// TIA Portal V17 program export: 1 tag tables, 0 data types, 18 data blocks, 11 code blocks (in call order from the OBs), 0 instance data blocks

VAR_GLOBAL   // PLC tag table "默认变量表"
   "1号计量泵运行" AT %I0.0 : Bool;
   "2号计量泵运行" AT %I0.2 : Bool;
   "3号计量泵运行" AT %I0.4 : Bool;
   "1号计量泵故障" AT %I0.1 : Bool;
   "2号计量泵故障" AT %I0.3 : Bool;
   "3号计量泵故障" AT %I0.5 : Bool;
   "1号药池电动阀开到位" AT %I0.6 : Bool;
   "2号药池电动阀开到位" AT %I1.0 : Bool;
   "1号药池电动阀关到位" AT %I0.7 : Bool;
   "2号药池电动阀关到位" AT %I1.1 : Bool;
   新旧电柜控制切换 AT %I1.2 : Bool;
   本电柜和中控控制切换 AT %I1.3 : Bool;
   "1号计量泵启停" AT %Q0.0 : Bool;
   "2号计量泵启停" AT %Q0.1 : Bool;
   "3号计量泵启停" AT %Q0.2 : Bool;
   "1号药池电动阀打开关闭" AT %Q0.3 : Bool;
   "2号药池电动阀打开关闭" AT %Q0.4 : Bool;
END_VAR

DATA_BLOCK "RS-485流量计1"
{ S7_Optimized_Access := 'FALSE' }
VERSION : 0.1
NON_RETAIN
   STRUCT 
      "40001" : Word;
      "40002" : Word;
      "40003" : Word;
      "40004" : Word;
      "40005" : Word;
      "40006" : Word;
      "40007" : Word;
      "40008" : Word;
      "40009" : Word;
      "40010" : Word;
      "40011" : Word;
      "40012" : Word;
      "40013" : Word;
      "40014" : Word;
      "40015" : Word;
      "40016" : Word;
      "40017" : Word;
      "40018" : Word;
      "40019" : Word;
      "40020" : Word;
      "40021" : Word;
      "40022" : Word;
      "40023" : Word;
      "40024" : Word;
      "40025" : Word;
      "40026" : Word;
      "40027" : Word;
      "40028" : Word;
      "40029" : Word;
      "40030" : Word;
      "40031" : Word;
      "40032" : Word;
      "40033" : Word;
      "40034" : Word;
      "40035" : Word;
      "40036" : Word;
      "40037" : Word;
      "40038" : Word;
      "40039" : Word;
      "40040" : Word;
      "40041" : Word;
      "40042" : Word;
      "40043" : Word;
      "40044" : Word;
      "40045" : Word;
      "40046" : Word;
      "40047" : Word;
      "40048" : Word;
      "40049" : Word;
      "40050" : Word;
   END_STRUCT;


BEGIN

END_DATA_BLOCK

DATA_BLOCK "RS-485流量计2"
{ S7_Optimized_Access := 'FALSE' }
VERSION : 0.1
NON_RETAIN
   STRUCT 
      "40001" : Word;
      "40002" : Word;
      "40003" : Word;
      "40004" : Word;
      "40005" : Word;
      "40006" : Word;
      "40007" : Word;
      "40008" : Word;
      "40009" : Word;
      "40010" : Word;
      "40011" : Word;
      "40012" : Word;
      "40013" : Word;
      "40014" : Word;
      "40015" : Word;
      "40016" : Word;
      "40017" : Word;
      "40018" : Word;
      "40019" : Word;
      "40020" : Word;
      "40021" : Word;
      "40022" : Word;
      "40023" : Word;
      "40024" : Word;
      "40025" : Word;
      "40026" : Word;
      "40027" : Word;
      "40028" : Word;
      "40029" : Word;
      "40030" : Word;
      "40031" : Word;
      "40032" : Word;
      "40033" : Word;
      "40034" : Word;
      "40035" : Word;
      "40036" : Word;
      "40037" : Word;
      "40038" : Word;
      "40039" : Word;
      "40040" : Word;
      "40041" : Word;
      "40042" : Word;
      "40043" : Word;
      "40044" : Word;
      "40045" : Word;
      "40046" : Word;
      "40047" : Word;
      "40048" : Word;
      "40049" : Word;
      "40050" : Word;
   END_STRUCT;


BEGIN

END_DATA_BLOCK

DATA_BLOCK "RS-485流量计3"
{ S7_Optimized_Access := 'FALSE' }
VERSION : 0.1
NON_RETAIN
   STRUCT 
      "40001" : Word;
      "40002" : Word;
      "40003" : Word;
      "40004" : Word;
      "40005" : Word;
      "40006" : Word;
      "40007" : Word;
      "40008" : Word;
      "40009" : Word;
      "40010" : Word;
      "40011" : Word;
      "40012" : Word;
      "40013" : Word;
      "40014" : Word;
      "40015" : Word;
      "40016" : Word;
      "40017" : Word;
      "40018" : Word;
      "40019" : Word;
      "40020" : Word;
      "40021" : Word;
      "40022" : Word;
      "40023" : Word;
      "40024" : Word;
      "40025" : Word;
      "40026" : Word;
      "40027" : Word;
      "40028" : Word;
      "40029" : Word;
      "40030" : Word;
      "40031" : Word;
      "40032" : Word;
      "40033" : Word;
      "40034" : Word;
      "40035" : Word;
      "40036" : Word;
      "40037" : Word;
      "40038" : Word;
      "40039" : Word;
      "40040" : Word;
      "40041" : Word;
      "40042" : Word;
      "40043" : Word;
      "40044" : Word;
      "40045" : Word;
      "40046" : Word;
      "40047" : Word;
      "40048" : Word;
      "40049" : Word;
      "40050" : Word;
   END_STRUCT;


BEGIN

END_DATA_BLOCK

DATA_BLOCK "RS-485电能表"
{ S7_Optimized_Access := 'FALSE' }
VERSION : 0.1
NON_RETAIN
   STRUCT 
      "40000" : Word;
      "40001" : Word;
      "40002" : Word;
      "40003" : Word;
      "40004" : Word;
      "40005" : Word;
      "40006" : Word;
      "40007" : Word;
      "40008" : Word;
      "40009" : Word;
      "40010" : Word;
      "40011" : Word;
      "40012" : Word;
      "40013" : Word;
      "40014" : Word;
      "40015" : Word;
      "40016" : Word;
      "40017" : Word;
      "40018" : Word;
      "40019" : Word;
      "40020" : Word;
      "40021" : Word;
      "40022" : Word;
      "40023" : Word;
      "40024" : Word;
      "40025" : Word;
      "40026" : Word;
      "40027" : Word;
      "40028" : Word;
      "40029" : Word;
      "40030" : Word;
      "40031" : Word;
      "40032" : Word;
      "40033" : Word;
      "40034" : Word;
      "40035" : Word;
      "40036" : Word;
      "40037" : Word;
      "40038" : Word;
      "40039" : Word;
      "40040" : Word;
      "40041" : Word;
      "40042" : Word;
      "40043" : Word;
      "40044" : Word;
      "40045" : Word;
      "40046" : Word;
      "40047" : Word;
      "40048" : Word;
      "40049" : Word;
      "40050" : Word;
      "40051" : Word;
      "40052" : Word;
      "40053" : Word;
      "40054" : Word;
      "40055" : Word;
      "40056" : Word;
      "40057" : Word;
      "40058" : Word;
      "40059" : Word;
      "40060" : Word;
      "40061" : Word;
      "40062" : Word;
      "40063" : Word;
      "40064" : Word;
      "40065" : Word;
      "40066" : Word;
      "40067" : Word;
      "40068" : Word;
      "40069" : Word;
      "40070" : Word;
      "40071" : Word;
      "40072" : Word;
      "40073" : Word;
      "40074" : Word;
      "40075" : Word;
      "40076" : Word;
      "40077" : Word;
      "40078" : Word;
   END_STRUCT;


BEGIN

END_DATA_BLOCK

DATA_BLOCK "local_control"
{ S7_Optimized_Access := 'FALSE' }
VERSION : 0.1
   STRUCT 
      start_stop : Array[0..5] of Bool;
      pump_maintain : Array[0..5] of Bool;
      flow_set : Array[0..5] of Real;
      flow_read : Array[0..5] of Real;
      tank_level : Array[0..5] of Real;
      valve_action : Array[0..5] of Bool;
      low_level_alarm : Array[0..5] of Bool;
      low_level_alarm_set : Array[0..5] of Real;
      flow_meter_read : Array[0..50] of Bool;
      flow_meter_read_error : Array[0..5] of Word;
      dosing_flow : Array[0..20] of Real;
      dosing_accumulate : Array[0..20] of Real;
      valve_opening : Array[0..5] of Bool;
      valve_closing : Array[0..5] of Bool;
      high_level_alarm : Array[0..5] of Bool;
      high_level_alarm_set : Array[0..5] of Real;
      energy_meter : Array[0..10] of Real;
      tank_weigh : Array[0..5] of Real;
      low_flow_alarm_set : Array[0..10] of Real;
      low_flow_alarm : Array[0..10] of Bool;
   END_STRUCT;


BEGIN

END_DATA_BLOCK

DATA_BLOCK "pump_local_control"
{ S7_Optimized_Access := 'TRUE' }
VERSION : 0.1
NON_RETAIN
   VAR 
      start_stop : Array[0..5] of Bool;
      pump_maintain : Array[0..5] of Bool;
      flow_set : Array[0..5] of Real;
   END_VAR


BEGIN

END_DATA_BLOCK

DATA_BLOCK "pump_remote_control"
{ S7_Optimized_Access := 'TRUE' }
VERSION : 0.1
NON_RETAIN
   VAR 
      start_stop : Array[0..5] of Bool;
      pump_maintain : Array[0..5] of Bool;
      flow_set : Array[0..5] of Real;
   END_VAR


BEGIN

END_DATA_BLOCK

DATA_BLOCK "pump_start_stop_DB1"
{ S7_Optimized_Access := 'TRUE' }
VERSION : 0.1
NON_RETAIN
"pump_start_stop"

BEGIN

END_DATA_BLOCK

DATA_BLOCK "pump_start_stop_DB2"
{ S7_Optimized_Access := 'TRUE' }
VERSION : 0.1
NON_RETAIN
"pump_start_stop"

BEGIN

END_DATA_BLOCK

DATA_BLOCK "pump_start_stop_DB3"
{ S7_Optimized_Access := 'TRUE' }
VERSION : 0.1
NON_RETAIN
"pump_start_stop"

BEGIN

END_DATA_BLOCK

DATA_BLOCK "pump_start_stop_DB4"
{ S7_Optimized_Access := 'TRUE' }
VERSION : 0.1
NON_RETAIN
"pump_start_stop"

BEGIN

END_DATA_BLOCK

DATA_BLOCK "pump_start_stop_DB5"
{ S7_Optimized_Access := 'TRUE' }
VERSION : 0.1
NON_RETAIN
"pump_start_stop"

BEGIN

END_DATA_BLOCK

DATA_BLOCK "pump_start_stop_DB6"
{ S7_Optimized_Access := 'TRUE' }
VERSION : 0.1
NON_RETAIN
"pump_start_stop"

BEGIN

END_DATA_BLOCK

DATA_BLOCK "RS-485"
{ S7_Optimized_Access := 'FALSE' }
VERSION : 0.1
NON_RETAIN
   STRUCT 
      "40001" : Word;
      "40002" : Word;
      "40003" : Word;
      "40004" : Word;
      "40005" : Word;
      "40006" : Word;
      "40007" : Word;
      "40008" : Word;
      "40009" : Word;
      "40010" : Word;
      "40011" : Word;
      "40012" : Word;
      "40013" : Word;
      "40014" : Word;
      "40015" : Word;
      "40016" : Word;
      "40017" : Word;
      "40018" : Word;
      "40019" : Word;
      "40020" : Word;
      "40021" : Word;
      "40022" : Word;
      "40023" : Word;
      "40024" : Word;
      "40025" : Word;
      "40026" : Word;
      "40027" : Word;
      "40028" : Word;
      "40029" : Word;
      "40030" : Word;
      "40031" : Word;
      "40032" : Word;
      "40033" : Word;
      "40034" : Word;
      "40035" : Word;
      "40036" : Word;
      "40037" : Word;
      "40038" : Word;
      "40039" : Word;
      "40040" : Word;
      "40041" : Word;
      "40042" : Word;
      "40043" : Word;
      "40044" : Word;
      "40045" : Word;
      "40046" : Word;
      "40047" : Word;
      "40048" : Word;
      "40049" : Word;
      "40050" : Word;
   END_STRUCT;


BEGIN

END_DATA_BLOCK

DATA_BLOCK "pump_flow_DB1"
{ S7_Optimized_Access := 'TRUE' }
VERSION : 0.1
NON_RETAIN
"pump_flow_set"

BEGIN

END_DATA_BLOCK

DATA_BLOCK "IEC_Timer_0_DB"
{InstructionName := 'IEC_TIMER';
 LibVersion := '1.0';
 S7_Optimized_Access := 'TRUE' }
AUTHOR : Simatic
FAMILY : IEC
NAME : IEC_TMR
VERSION : 1.0
NON_RETAIN
IEC_TIMER

BEGIN

END_DATA_BLOCK

DATA_BLOCK "MB_COMM_LOAD_DB"
{InstructionName := 'MB_COMM_LOAD';
 LibVersion := '2.1';
 S7_Optimized_Access := 'TRUE' }
AUTHOR : SIMATIC
FAMILY : MODBUS
NAME : MB_CM_LD
VERSION : 2.1
NON_RETAIN
MB_COMM_LOAD

BEGIN

END_DATA_BLOCK

DATA_BLOCK "MB_MASTER_DB"
{InstructionName := 'MB_MASTER';
 LibVersion := '2.2';
 S7_Optimized_Access := 'TRUE' }
AUTHOR : SIMATIC
FAMILY : MODBUS
NAME : MB_MASTR
VERSION : 2.2
NON_RETAIN
MB_MASTER

BEGIN

END_DATA_BLOCK

ORGANIZATION_BLOCK "Main"   // OB1, LAD, ProgramCycle
TITLE = "Main Program Sweep (Cycle)"
{ S7_Optimized_Access := 'TRUE' }
VERSION : 0.1
// stored: AutoNumber true, IsIECCheckEnabled false, SetENOAutomatically false
   VAR_INPUT
      Initial_Call : Bool;   // Initial call of this OB
      Remanence : Bool;   // =True, if remanent data are available
   END_VAR
BEGIN

REGION Network 1
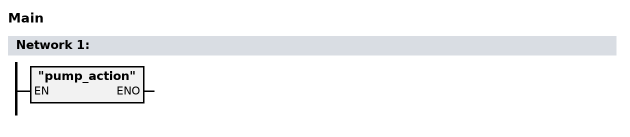
   RUNG wire#powerrail
      "pump_action"()
   END_RUNG
   // the same network as SCL:
   "pump_action"();
END_REGION
END_ORGANIZATION_BLOCK

FUNCTION "pump_action" : Void   // FC1, LAD
{ S7_Optimized_Access := 'TRUE' }
VERSION : 0.1
// stored: AutoNumber true, IsIECCheckEnabled false, SetENOAutomatically false, UDAEnableTagReadback false
BEGIN

REGION Network 1
   // 1号泵
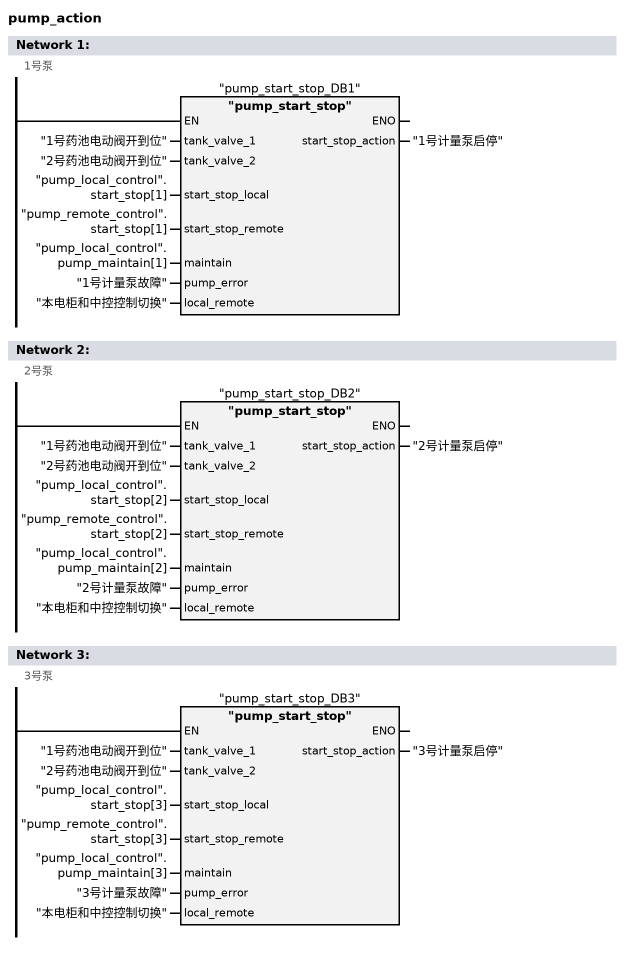
   RUNG wire#powerrail
      "pump_start_stop_DB1"(tank_valve_1 := "1号药池电动阀开到位", tank_valve_2 := "2号药池电动阀开到位", start_stop_local := "pump_local_control".start_stop[1], start_stop_remote := "pump_remote_control".start_stop[1], maintain := "pump_local_control".pump_maintain[1], pump_error := "1号计量泵故障", local_remote := "本电柜和中控控制切换", start_stop_action => "1号计量泵启停")
   END_RUNG
   // the same network as SCL:
   "pump_start_stop_DB1"(tank_valve_1 := "1号药池电动阀开到位",   // "pump_start_stop"
                         tank_valve_2 := "2号药池电动阀开到位",
                         start_stop_local := "pump_local_control".start_stop[1],
                         start_stop_remote := "pump_remote_control".start_stop[1],
                         maintain := "pump_local_control".pump_maintain[1],
                         pump_error := "1号计量泵故障",
                         local_remote := "本电柜和中控控制切换",
                         start_stop_action => "1号计量泵启停");
END_REGION

REGION Network 2
   // 2号泵
   RUNG wire#powerrail
      "pump_start_stop_DB2"(tank_valve_1 := "1号药池电动阀开到位", tank_valve_2 := "2号药池电动阀开到位", start_stop_local := "pump_local_control".start_stop[2], start_stop_remote := "pump_remote_control".start_stop[2], maintain := "pump_local_control".pump_maintain[2], pump_error := "2号计量泵故障", local_remote := "本电柜和中控控制切换", start_stop_action => "2号计量泵启停")
   END_RUNG
   // the same network as SCL:
   "pump_start_stop_DB2"(tank_valve_1 := "1号药池电动阀开到位",   // "pump_start_stop"
                         tank_valve_2 := "2号药池电动阀开到位",
                         start_stop_local := "pump_local_control".start_stop[2],
                         start_stop_remote := "pump_remote_control".start_stop[2],
                         maintain := "pump_local_control".pump_maintain[2],
                         pump_error := "2号计量泵故障",
                         local_remote := "本电柜和中控控制切换",
                         start_stop_action => "2号计量泵启停");
END_REGION

REGION Network 3
   // 3号泵
   RUNG wire#powerrail
      "pump_start_stop_DB3"(tank_valve_1 := "1号药池电动阀开到位", tank_valve_2 := "2号药池电动阀开到位", start_stop_local := "pump_local_control".start_stop[3], start_stop_remote := "pump_remote_control".start_stop[3], maintain := "pump_local_control".pump_maintain[3], pump_error := "3号计量泵故障", local_remote := "本电柜和中控控制切换", start_stop_action => "3号计量泵启停")
   END_RUNG
   // the same network as SCL:
   "pump_start_stop_DB3"(tank_valve_1 := "1号药池电动阀开到位",   // "pump_start_stop"
                         tank_valve_2 := "2号药池电动阀开到位",
                         start_stop_local := "pump_local_control".start_stop[3],
                         start_stop_remote := "pump_remote_control".start_stop[3],
                         maintain := "pump_local_control".pump_maintain[3],
                         pump_error := "3号计量泵故障",
                         local_remote := "本电柜和中控控制切换",
                         start_stop_action => "3号计量泵启停");
END_REGION
END_FUNCTION

FUNCTION_BLOCK "pump_start_stop"   // FB1, LAD
{ S7_Optimized_Access := 'TRUE' }
VERSION : 0.1
// stored: AutoNumber true, IsIECCheckEnabled false, IsRetainMemResEnabled false, MemoryReserve 100, SetENOAutomatically false, UDAEnableTagReadback false
   VAR_INPUT
      tank_valve_1 : Bool;
      tank_valve_2 : Bool;
      start_stop_local : Bool;
      start_stop_remote : Bool;
      maintain : Bool;
      pump_error : Bool;
      local_remote : Bool;
   END_VAR
   VAR_OUTPUT
      start_stop_action : Bool;
   END_VAR
BEGIN

REGION Network 1
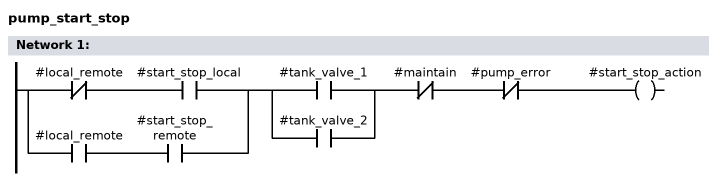
   RUNG wire#powerrail
      I_Contact( #local_remote )
      Contact( #start_stop_local )
      wire#w1
      Contact( #tank_valve_1 )
      wire#w2
      I_Contact( #maintain )
      I_Contact( #pump_error )
      Coil( #start_stop_action )
   END_RUNG
   RUNG wire#powerrail
      Contact( #local_remote )
      Contact( #start_stop_remote )
   END_RUNG wire#w1
   RUNG wire#w1
      Contact( #tank_valve_2 )
   END_RUNG wire#w2
   // the same network as SCL:
   #start_stop_action := ((NOT #local_remote AND #start_stop_local) OR (#local_remote AND #start_stop_remote)) AND (#tank_valve_1 OR #tank_valve_2) AND NOT #maintain AND NOT #pump_error;
END_REGION
END_FUNCTION_BLOCK

ORGANIZATION_BLOCK "Startup"   // OB100, LAD, Startup
TITLE = "Complete Restart"
{ S7_Optimized_Access := 'TRUE' }
VERSION : 0.1
// stored: AutoNumber true, IsIECCheckEnabled false, SetENOAutomatically false
   VAR_INPUT
      LostRetentive : Bool;   // True if retentive data are lost
      LostRTC : Bool;   // True if date and time are lost
   END_VAR
BEGIN

REGION Network 1
   // 建立RS-485连接
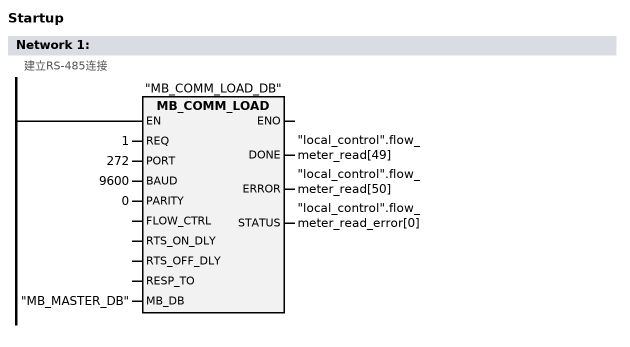
   RUNG wire#powerrail
      "MB_COMM_LOAD_DB".MB_COMM_LOAD(REQ := 1, PORT := 272, BAUD := 9600, PARITY := 0, FLOW_CTRL :=, RTS_ON_DLY :=, RTS_OFF_DLY :=, RESP_TO :=, MB_DB := "MB_MASTER_DB", DONE => "local_control".flow_meter_read[49], ERROR => "local_control".flow_meter_read[50], STATUS => "local_control".flow_meter_read_error[0])
   END_RUNG
   // the same network as SCL:
   "MB_COMM_LOAD_DB"(REQ := 1,   // MB_COMM_LOAD
                     PORT := 272,
                     BAUD := 9600,
                     PARITY := 0,
                     MB_DB := "MB_MASTER_DB",
                     DONE => "local_control".flow_meter_read[49],
                     ERROR => "local_control".flow_meter_read[50],
                     STATUS => "local_control".flow_meter_read_error[0]);
END_REGION
END_ORGANIZATION_BLOCK

FUNCTION "energy_meter_read" : Void   // FC7, SCL
{ S7_Optimized_Access := 'TRUE' }
VERSION : 0.1
// stored: AutoNumber true, IsIECCheckEnabled false, SetENOAutomatically false, UDAEnableTagReadback false
BEGIN
   //读电能表数据

   //读电压
   //A相
   %DB2. := %DB5.;
   %DB2. := %DB5.;
   "local_control".energy_meter[0] := "local_control".energy_meter[0] / 10.0;

   //读电压
   //B相
   %DB2. := %DB5.;
   %DB2. := %DB5.;
   "local_control".energy_meter[1] := "local_control".energy_meter[1] / 10.0;

   //读电压
   //C相
   %DB2. := %DB5.;
   %DB2. := %DB5.;
   "local_control".energy_meter[2] := "local_control".energy_meter[2] / 10.0;

   //读电流
   //A相
   %DB2. := %DB5.;
   %DB2. := %DB5.;
   "local_control".energy_meter[3] := "local_control".energy_meter[3] / 1000.0;

   //读电流
   //B相
   %DB2. := %DB5.;
   %DB2. := %DB5.;
   "local_control".energy_meter[4] := "local_control".energy_meter[4] / 1000.0;

   //读电流
   //C相
   %DB2. := %DB5.;
   %DB2. := %DB5.;
   "local_control".energy_meter[5] := "local_control".energy_meter[5] / 1000.0;

   //读电能
   //正向有功总电能
   %DB2. := %DB5.;
   %DB2. := %DB5.;
   "local_control".energy_meter[6] := "local_control".energy_meter[6] / 10.0;
END_FUNCTION

FUNCTION "RS-485_connect" : Void   // FC5, LAD
{ S7_Optimized_Access := 'TRUE' }
VERSION : 0.1
// stored: AutoNumber true, IsIECCheckEnabled false, SetENOAutomatically false, UDAEnableTagReadback false
   VAR_TEMP   // added for the SCL form of the ladder/FBD networks
      _w1 : Bool;
      _w2 : Bool;
      _w3 : Bool;
      _w4 : Bool;
      _w5 : Bool;
   END_VAR
BEGIN

REGION Network 1: 读从站
   // 读流量计从站
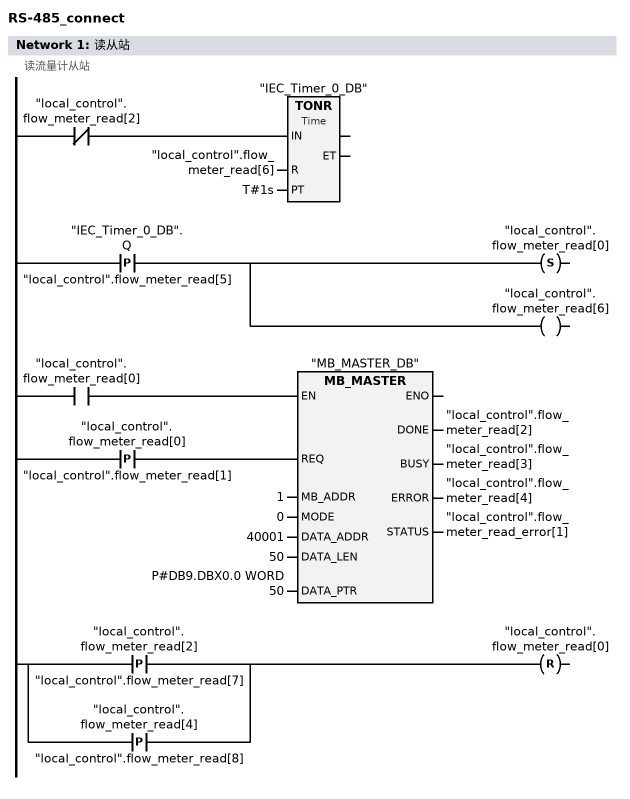
   RUNG wire#powerrail
      I_Contact( "local_control".flow_meter_read[2] )
      { S7_Templates := "time_type := Time" } "IEC_Timer_0_DB".TONR(r := "local_control".flow_meter_read[6], pt := T#1s, et =>)
   END_RUNG
   RUNG wire#powerrail
      P_Contact(operand := "IEC_Timer_0_DB".Q, bit := "local_control".flow_meter_read[5])
      wire#w1
      S_Coil( "local_control".flow_meter_read[0] )
   END_RUNG
   RUNG wire#w1
      Coil( "local_control".flow_meter_read[6] )
   END_RUNG
   RUNG wire#powerrail
      Contact( "local_control".flow_meter_read[0] )
      "MB_MASTER_DB".MB_MASTER(REQ := wire#w2, MB_ADDR := 1, MODE := 0, DATA_ADDR := 40001, DATA_LEN := 50, DATA_PTR := P#DB9.DBX0.0 WORD 50, DONE => "local_control".flow_meter_read[2], BUSY => "local_control".flow_meter_read[3], ERROR => "local_control".flow_meter_read[4], STATUS => "local_control".flow_meter_read_error[1])
   END_RUNG
   RUNG wire#powerrail
      P_Contact(operand := "local_control".flow_meter_read[0], bit := "local_control".flow_meter_read[1])
   END_RUNG wire#w2
   RUNG wire#powerrail
      P_Contact(operand := "local_control".flow_meter_read[2], bit := "local_control".flow_meter_read[7])
      wire#w3
      R_Coil( "local_control".flow_meter_read[0] )
   END_RUNG
   RUNG wire#powerrail
      P_Contact(operand := "local_control".flow_meter_read[4], bit := "local_control".flow_meter_read[8])
   END_RUNG wire#w3
   // the same network as SCL:
   "IEC_Timer_0_DB".TONR(IN := NOT "local_control".flow_meter_read[2],
                         R := "local_control".flow_meter_read[6],
                         PT := T#1s);
   #_w1 := "IEC_Timer_0_DB".Q AND NOT "local_control".flow_meter_read[5];   // rising edge of "IEC_Timer_0_DB".Q
   "local_control".flow_meter_read[5] := "IEC_Timer_0_DB".Q;
   IF #_w1 THEN "local_control".flow_meter_read[0] := TRUE; END_IF;
   "local_control".flow_meter_read[6] := #_w1;
   #_w3 := "local_control".flow_meter_read[0];
   #_w2 := "local_control".flow_meter_read[0] AND NOT "local_control".flow_meter_read[1];   // rising edge of "local_control".flow_meter_read[0]
   "local_control".flow_meter_read[1] := "local_control".flow_meter_read[0];
   IF #_w3 THEN
       "MB_MASTER_DB"(REQ := #_w2,   // MB_MASTER
                      MB_ADDR := 1,
                      MODE := 0,
                      DATA_ADDR := 40001,
                      DATA_LEN := 50,
                      DATA_PTR := P#DB9.DBX0.0 WORD 50,
                      DONE => "local_control".flow_meter_read[2],
                      BUSY => "local_control".flow_meter_read[3],
                      ERROR => "local_control".flow_meter_read[4],
                      STATUS => "local_control".flow_meter_read_error[1]);
   END_IF;
   #_w4 := "local_control".flow_meter_read[2] AND NOT "local_control".flow_meter_read[7];   // rising edge of "local_control".flow_meter_read[2]
   "local_control".flow_meter_read[7] := "local_control".flow_meter_read[2];
   #_w5 := "local_control".flow_meter_read[4] AND NOT "local_control".flow_meter_read[8];   // rising edge of "local_control".flow_meter_read[4]
   "local_control".flow_meter_read[8] := "local_control".flow_meter_read[4];
   IF #_w4 OR #_w5 THEN "local_control".flow_meter_read[0] := FALSE; END_IF;
END_REGION
END_FUNCTION

FUNCTION_BLOCK "pump_flow_set"   // FB2, LAD
{ S7_Optimized_Access := 'TRUE' }
VERSION : 0.1
// stored: AutoNumber true, IsIECCheckEnabled false, IsRetainMemResEnabled false, MemoryReserve 100, SetENOAutomatically false, UDAEnableTagReadback false
   VAR_INPUT
      local_remote : Bool;
      local_flow_set : Real;
      remote_flow_set : Real;
   END_VAR
   VAR_OUTPUT
      flow_set_output : Real;
   END_VAR
   VAR_TEMP
      control_flow : Real;
      flow_temp_real : Real;
   END_VAR
BEGIN

REGION Network 1
   // 远程/在地切换
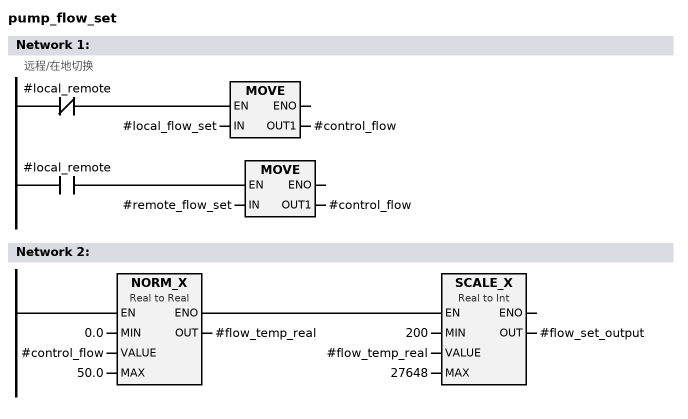
   RUNG wire#powerrail
      I_Contact( #local_remote )
      Move(in := #local_flow_set, out1 => #control_flow)
   END_RUNG
   RUNG wire#powerrail
      Contact( #local_remote )
      Move(in := #remote_flow_set, out1 => #control_flow)
   END_RUNG
   // the same network as SCL:
   IF NOT #local_remote THEN #control_flow := #local_flow_set; END_IF;
   IF #local_remote THEN #control_flow := #remote_flow_set; END_IF;
END_REGION

REGION Network 2
   RUNG wire#powerrail
      { S7_Templates := "[SrcType := Real, DestType := Real]" } Normalize(min := 0.0, value := #control_flow, max := 50.0, out => #flow_temp_real)
      { S7_Templates := "[SrcType := Real, DestType := Int]" } Scale(min := 200, value := #flow_temp_real, max := 27648, out => #flow_set_output)
   END_RUNG
   // the same network as SCL:
   #flow_temp_real := NORM_X(MIN := 0.0, VALUE := #control_flow, MAX := 50.0);
   #flow_set_output := SCALE_X(MIN := 200, VALUE := #flow_temp_real, MAX := 27648);
END_REGION
END_FUNCTION_BLOCK

FUNCTION "pump_flow_set_and_read" : Void   // FC2, LAD
{ S7_Optimized_Access := 'TRUE' }
VERSION : 0.1
// stored: AutoNumber true, IsIECCheckEnabled false, SetENOAutomatically false, UDAEnableTagReadback false
   VAR_TEMP
      flow_read_temp1 : Real;
      flow_read_temp2 : Real;
      flow_read_temp3 : Real;
   END_VAR
BEGIN

REGION Network 1
   // 1号泵流量控制
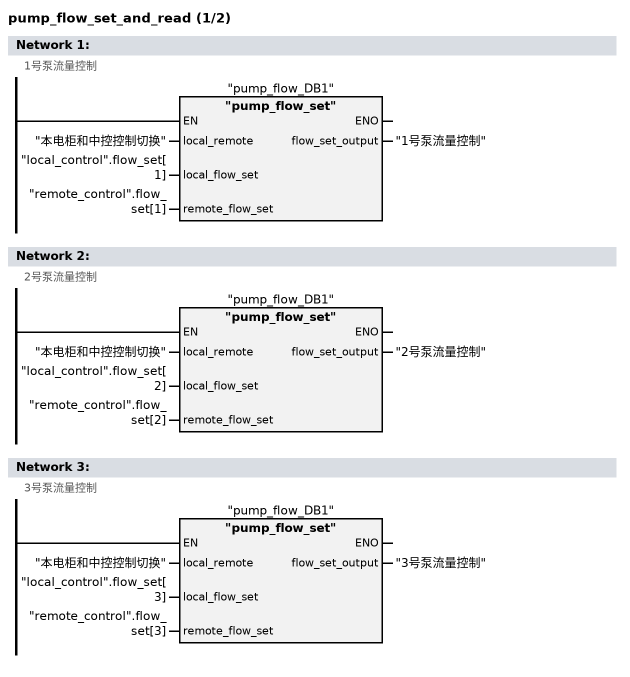
   RUNG wire#powerrail
      "pump_flow_DB1"(local_remote := "本电柜和中控控制切换", local_flow_set := "local_control".flow_set[1], remote_flow_set := "remote_control".flow_set[1], flow_set_output => "1号泵流量控制")
   END_RUNG
   // the same network as SCL:
   "pump_flow_DB1"(local_remote := "本电柜和中控控制切换",   // "pump_flow_set"
                   local_flow_set := "local_control".flow_set[1],
                   remote_flow_set := "remote_control".flow_set[1],
                   flow_set_output => "1号泵流量控制");
END_REGION

REGION Network 2
   // 2号泵流量控制
   RUNG wire#powerrail
      "pump_flow_DB1"(local_remote := "本电柜和中控控制切换", local_flow_set := "local_control".flow_set[2], remote_flow_set := "remote_control".flow_set[2], flow_set_output => "2号泵流量控制")
   END_RUNG
   // the same network as SCL:
   "pump_flow_DB1"(local_remote := "本电柜和中控控制切换",   // "pump_flow_set"
                   local_flow_set := "local_control".flow_set[2],
                   remote_flow_set := "remote_control".flow_set[2],
                   flow_set_output => "2号泵流量控制");
END_REGION

REGION Network 3
   // 3号泵流量控制
   RUNG wire#powerrail
      "pump_flow_DB1"(local_remote := "本电柜和中控控制切换", local_flow_set := "local_control".flow_set[3], remote_flow_set := "remote_control".flow_set[3], flow_set_output => "3号泵流量控制")
   END_RUNG
   // the same network as SCL:
   "pump_flow_DB1"(local_remote := "本电柜和中控控制切换",   // "pump_flow_set"
                   local_flow_set := "local_control".flow_set[3],
                   remote_flow_set := "remote_control".flow_set[3],
                   flow_set_output => "3号泵流量控制");
END_REGION

REGION Network 4
   // 读取计量泵反馈流量
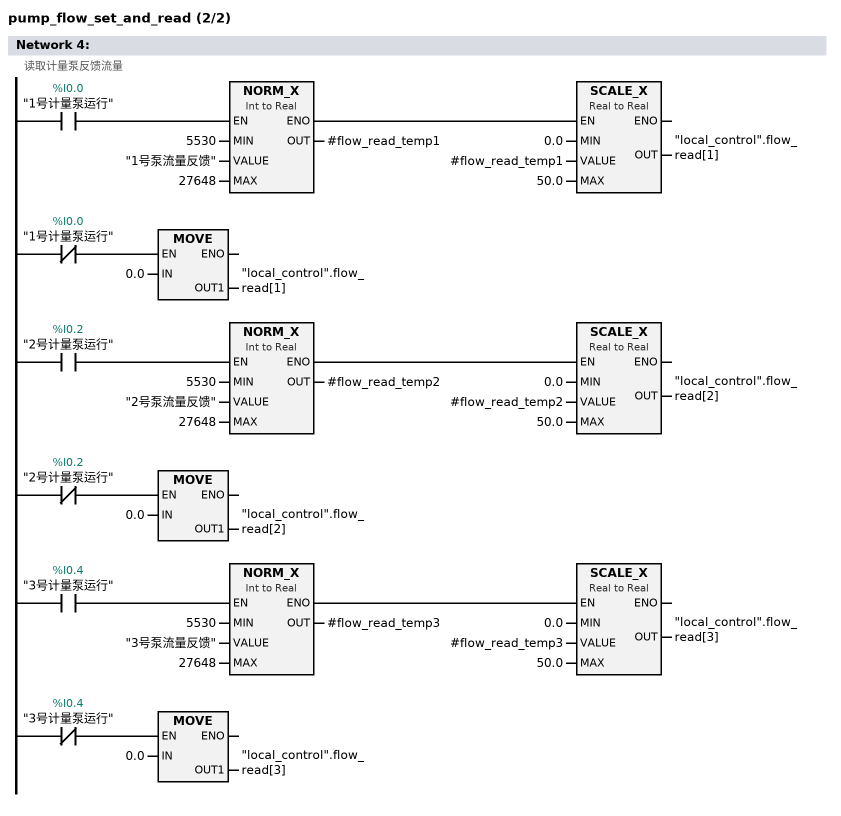
   RUNG wire#powerrail
      Contact( "1号计量泵运行" )
      { S7_Templates := "[SrcType := Int, DestType := Real]" } Normalize(min := 5530, value := "1号泵流量反馈", max := 27648, out => #flow_read_temp1)
      { S7_Templates := "[SrcType := Real, DestType := Real]" } Scale(min := 0.0, value := #flow_read_temp1, max := 50.0, out => "local_control".flow_read[1])
   END_RUNG
   RUNG wire#powerrail
      I_Contact( "1号计量泵运行" )
      Move(in := 0.0, out1 => "local_control".flow_read[1])
   END_RUNG
   RUNG wire#powerrail
      Contact( "2号计量泵运行" )
      { S7_Templates := "[SrcType := Int, DestType := Real]" } Normalize(min := 5530, value := "2号泵流量反馈", max := 27648, out => #flow_read_temp2)
      { S7_Templates := "[SrcType := Real, DestType := Real]" } Scale(min := 0.0, value := #flow_read_temp2, max := 50.0, out => "local_control".flow_read[2])
   END_RUNG
   RUNG wire#powerrail
      I_Contact( "2号计量泵运行" )
      Move(in := 0.0, out1 => "local_control".flow_read[2])
   END_RUNG
   RUNG wire#powerrail
      Contact( "3号计量泵运行" )
      { S7_Templates := "[SrcType := Int, DestType := Real]" } Normalize(min := 5530, value := "3号泵流量反馈", max := 27648, out => #flow_read_temp3)
      { S7_Templates := "[SrcType := Real, DestType := Real]" } Scale(min := 0.0, value := #flow_read_temp3, max := 50.0, out => "local_control".flow_read[3])
   END_RUNG
   RUNG wire#powerrail
      I_Contact( "3号计量泵运行" )
      Move(in := 0.0, out1 => "local_control".flow_read[3])
   END_RUNG
   // the same network as SCL:
   IF "1号计量泵运行" THEN
       #flow_read_temp1 := NORM_X(MIN := 5530, VALUE := "1号泵流量反馈", MAX := 27648);
       "local_control".flow_read[1] := SCALE_X(MIN := 0.0, VALUE := #flow_read_temp1, MAX := 50.0);
   END_IF;
   IF NOT "1号计量泵运行" THEN "local_control".flow_read[1] := 0.0; END_IF;
   IF "2号计量泵运行" THEN
       #flow_read_temp2 := NORM_X(MIN := 5530, VALUE := "2号泵流量反馈", MAX := 27648);
       "local_control".flow_read[2] := SCALE_X(MIN := 0.0, VALUE := #flow_read_temp2, MAX := 50.0);
   END_IF;
   IF NOT "2号计量泵运行" THEN "local_control".flow_read[2] := 0.0; END_IF;
   IF "3号计量泵运行" THEN
       #flow_read_temp3 := NORM_X(MIN := 5530, VALUE := "3号泵流量反馈", MAX := 27648);
       "local_control".flow_read[3] := SCALE_X(MIN := 0.0, VALUE := #flow_read_temp3, MAX := 50.0);
   END_IF;
   IF NOT "3号计量泵运行" THEN "local_control".flow_read[3] := 0.0; END_IF;
END_REGION
END_FUNCTION

FUNCTION "tank_level" : Void   // FC3, LAD
{ S7_Optimized_Access := 'TRUE' }
VERSION : 0.1
// stored: AutoNumber true, IsIECCheckEnabled false, SetENOAutomatically false, UDAEnableTagReadback false
   VAR_TEMP
      tank_level_temp1 : Real;
      tank_level_temp2 : Real;
   END_VAR
BEGIN

REGION Network 1
   // 读取罐液罐液位
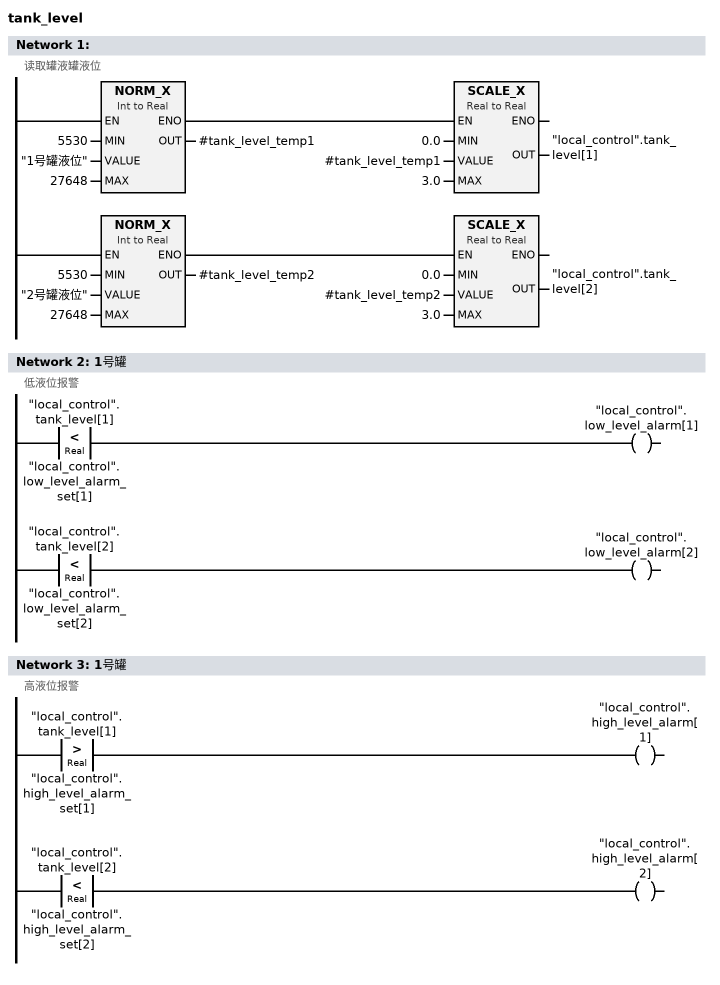
   RUNG wire#powerrail
      { S7_Templates := "[SrcType := Int, DestType := Real]" } Normalize(min := 5530, value := "1号罐液位", max := 27648, out => #tank_level_temp1)
      { S7_Templates := "[SrcType := Real, DestType := Real]" } Scale(min := 0.0, value := #tank_level_temp1, max := 3.0, out => "local_control".tank_level[1])
   END_RUNG
   RUNG wire#powerrail
      { S7_Templates := "[SrcType := Int, DestType := Real]" } Normalize(min := 5530, value := "2号罐液位", max := 27648, out => #tank_level_temp2)
      { S7_Templates := "[SrcType := Real, DestType := Real]" } Scale(min := 0.0, value := #tank_level_temp2, max := 3.0, out => "local_control".tank_level[2])
   END_RUNG
   // the same network as SCL:
   #tank_level_temp1 := NORM_X(MIN := 5530, VALUE := "1号罐液位", MAX := 27648);
   "local_control".tank_level[1] := SCALE_X(MIN := 0.0, VALUE := #tank_level_temp1, MAX := 3.0);
   #tank_level_temp2 := NORM_X(MIN := 5530, VALUE := "2号罐液位", MAX := 27648);
   "local_control".tank_level[2] := SCALE_X(MIN := 0.0, VALUE := #tank_level_temp2, MAX := 3.0);
END_REGION

REGION Network 2: 1号罐
   // 低液位报警
   RUNG wire#powerrail
      { S7_Templates := "SrcType := Real" } LT_Contact(in1 := "local_control".tank_level[1], in2 := "local_control".low_level_alarm_set[1])
      Coil( "local_control".low_level_alarm[1] )
   END_RUNG
   RUNG wire#powerrail
      { S7_Templates := "SrcType := Real" } LT_Contact(in1 := "local_control".tank_level[2], in2 := "local_control".low_level_alarm_set[2])
      Coil( "local_control".low_level_alarm[2] )
   END_RUNG
   // the same network as SCL:
   "local_control".low_level_alarm[1] := "local_control".tank_level[1] < "local_control".low_level_alarm_set[1];
   "local_control".low_level_alarm[2] := "local_control".tank_level[2] < "local_control".low_level_alarm_set[2];
END_REGION

REGION Network 3: 1号罐
   // 高液位报警
   RUNG wire#powerrail
      { S7_Templates := "SrcType := Real" } GT_Contact(in1 := "local_control".tank_level[1], in2 := "local_control".high_level_alarm_set[1])
      Coil( "local_control".high_level_alarm[1] )
   END_RUNG
   RUNG wire#powerrail
      { S7_Templates := "SrcType := Real" } LT_Contact(in1 := "local_control".tank_level[2], in2 := "local_control".high_level_alarm_set[2])
      Coil( "local_control".high_level_alarm[2] )
   END_RUNG
   // the same network as SCL:
   "local_control".high_level_alarm[1] := "local_control".tank_level[1] > "local_control".high_level_alarm_set[1];
   "local_control".high_level_alarm[2] := "local_control".tank_level[2] < "local_control".high_level_alarm_set[2];
END_REGION
END_FUNCTION

FUNCTION "valve_control" : Void   // FC4, LAD
{ S7_Optimized_Access := 'TRUE' }
VERSION : 0.1
// stored: AutoNumber true, IsIECCheckEnabled false, SetENOAutomatically false, UDAEnableTagReadback false
BEGIN

REGION Network 1
   // 1号电动阀
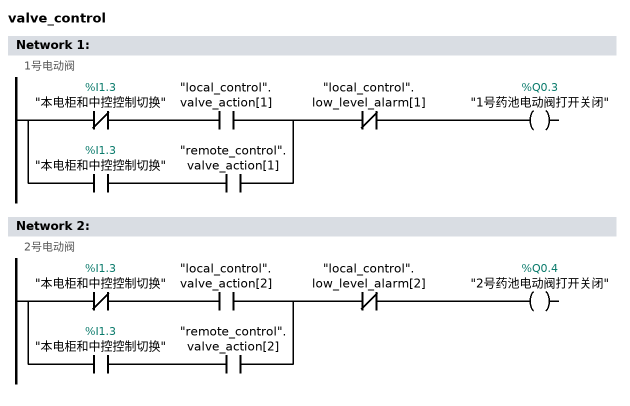
   RUNG wire#powerrail
      I_Contact( "本电柜和中控控制切换" )
      Contact( "local_control".valve_action[1] )
      wire#w1
      I_Contact( "local_control".low_level_alarm[1] )
      Coil( "1号药池电动阀打开关闭" )
   END_RUNG
   RUNG wire#powerrail
      Contact( "本电柜和中控控制切换" )
      Contact( "remote_control".valve_action[1] )
   END_RUNG wire#w1
   // the same network as SCL:
   "1号药池电动阀打开关闭" := ((NOT "本电柜和中控控制切换" AND "local_control".valve_action[1]) OR ("本电柜和中控控制切换" AND "remote_control".valve_action[1])) AND NOT "local_control".low_level_alarm[1];
END_REGION

REGION Network 2
   // 2号电动阀
   RUNG wire#powerrail
      I_Contact( "本电柜和中控控制切换" )
      Contact( "local_control".valve_action[2] )
      wire#w1
      I_Contact( "local_control".low_level_alarm[2] )
      Coil( "2号药池电动阀打开关闭" )
   END_RUNG
   RUNG wire#powerrail
      Contact( "本电柜和中控控制切换" )
      Contact( "remote_control".valve_action[2] )
   END_RUNG wire#w1
   // the same network as SCL:
   "2号药池电动阀打开关闭" := ((NOT "本电柜和中控控制切换" AND "local_control".valve_action[2]) OR ("本电柜和中控控制切换" AND "remote_control".valve_action[2])) AND NOT "local_control".low_level_alarm[2];
END_REGION
END_FUNCTION

FUNCTION "flow_meter_read" : Void
{ S7_Optimized_Access := 'TRUE' }
VERSION : 0.1

BEGIN
	//读流量仪表数据
	
	//瞬时流量
	//次氯酸钠
	"local_control".dosing_flow[1] := UINT_TO_REAL("RS-485"."40005")*32768.0 + UINT_TO_REAL("RS-485"."40006") +UINT_TO_REAL("RS-485"."40007") / 1000;
	"local_control".dosing_flow[2] := UINT_TO_REAL("RS-485"."40008") * 32768.0 + UINT_TO_REAL("RS-485"."40009") + UINT_TO_REAL("RS-485"."40010") / 1000;
	
	//累积容积
	//次氯酸钠
	"local_control".dosing_accumulate[1] := UINT_TO_REAL("RS-485"."40011") * 32768.0 ** 3.0 + UINT_TO_REAL("RS-485"."40012") * 32768.0 ** 2.0 + UINT_TO_REAL("RS-485"."40013") * 32768.0
	+ UINT_TO_REAL("RS-485"."40014")+ UINT_TO_REAL("RS-485"."40015") / 1000;
	"local_control".dosing_accumulate[2] := UINT_TO_REAL("RS-485"."40016") * 32768.0 ** 3.0 + UINT_TO_REAL("RS-485"."40017") * 32768.0 ** 2.0 + UINT_TO_REAL("RS-485"."40018") * 32768.0
	+ UINT_TO_REAL("RS-485"."40019") + UINT_TO_REAL("RS-485"."40020") / 1000;
END_FUNCTION
